TYPE T_Ctrl_SIf_FOL_Out :
STRUCT
END_STRUCT
END_TYPE

(* stored: Version 1.1.0.1, ProductVersion 3.1.0.19
   DUT T_Ctrl_SIf_FOL_Out: Id {27969bf5-2fb0-4b4f-93f3-56d11b0a6e18} *)
